{attribute addProperty BoxType "EL6201-0000-0017"}
{attribute addProperty Id "Slave_20A_DI0BIT10.125153Slave_20A_DI1BIT10.125154Slave_20A_DI2BIT10.125155Slave_20A_DI3BIT10.125156Slave_20B_DI0BIT10.125157Slave_20B_DI1BIT10.125158Slave_20B_DI2BIT10.125159Slave_20B_DI3BIT10.125160"}
{attribute addProperty CRC "2408740647"}
{attribute addProperty SizeInBites "8"}
{attribute addProperty SizeInBytes "1"}
TYPE Slave_20_Inputs_8F927727 :
STRUCT
	{attribute addProperty Name "Slave_20A_DI0"}
	Slave_20A_DI0 : BIT;
	{attribute addProperty Name "Slave_20A_DI1"}
	Slave_20A_DI1 : BIT;
	{attribute addProperty Name "Slave_20A_DI2"}
	Slave_20A_DI2 : BIT;
	{attribute addProperty Name "Slave_20A_DI3"}
	Slave_20A_DI3 : BIT;
	{attribute addProperty Name "Slave_20B_DI0"}
	Slave_20B_DI0 : BIT;
	{attribute addProperty Name "Slave_20B_DI1"}
	Slave_20B_DI1 : BIT;
	{attribute addProperty Name "Slave_20B_DI2"}
	Slave_20B_DI2 : BIT;
	{attribute addProperty Name "Slave_20B_DI3"}
	Slave_20B_DI3 : BIT;
END_STRUCT
END_TYPE

(* stored: Version 1.2.0.0, ProductVersion 3.1.4024.9
   DUT Slave_20_Inputs_8F927727: Id {c93a5ec5-1ea4-4cd4-b382-0694b9f0b466} *)
